// Implicitly generated code : DO NOT EDIT
FUNCTION CheckRangeUnsigned : UDINT
VAR_INPUT
	value, lower, upper: UDINT;
END_VAR

// Implicitly generated code : Only an Implementation suggestion
{noflow}
IF (value < lower) THEN
	CheckRangeUnsigned := lower;
	G_Diag.uiCheckRange:=G_Diag.uiCheckRange+1;
ELSIF(value > upper) THEN
	CheckRangeUnsigned := upper;
	G_Diag.uiCheckRange:=G_Diag.uiCheckRange+1;
ELSE
	CheckRangeUnsigned := value;
END_IF
{flow}

END_FUNCTION

(* stored: Version 1.1.0.1, ProductVersion 3.1.4024.4
   POU CheckRangeUnsigned: Id {8e82ee73-accb-49b8-8e55-f38f1b907d38}, SpecialFunc CheckRangeUnsigned *)
